Fanuc KAREL source: kt00062.KL

-- PROVISIONAL review KL for V770-1; original PC SHA256 1210aa0f38b67f4dec61d9eb6c73eddb2501100a545b9f9c89a4c6679023fff8
-- Incomplete behavior may be omitted. Consult companion uncertainty JSON. Do not deploy.
PROGRAM KT00062
%NOLOCKGROUP
VAR
  OUT : REAL
-- UNRESOLVED_DECL H1 type=002017
-- UNRESOLVED_DECL Y2 type=002018
BEGIN
  -- UNRESOLVED_PC offsets 5-19; opcodes 2E,22,9D,33,B4
  -- UNRESOLVED_PC offsets 24-38; opcodes 2E,22,9D,33,B2
  -- UNRESOLVED_PC offsets 43-69; opcodes 22,9D,33,B3,22,9D,33,B1,53,64,23
  -- UNRESOLVED_PC offsets 74-78; opcodes 7F
END KT00062
